// SIMATIC STEP 7 (V5.x) project Water tank
// CPU: CPU 413-2 DP
// station: Hardware
// station: SIMATIC 400(1)
// station: P_ADR_BUS
// station: P_ADR_BUS
// station: P_ADR_BUS
// station: Configuration
// program: S7 Program(1)

SYMBOL_TABLE
"Data For Temp"	DB 1	DB 1
"Temperature scaling"	FC 1	FC 1
"Motor operation"	FC 2	FC 2
"SCALE"	FC 105	FC 105	// Scaling Values
"Temp scaling"	OB 1	OB 1
"Tank-1"	PIW 256	INT	// temp for tank-1
"Tank-2"	PIW 258	INT	// temp for tank-2
"Temp-2"	PIW 512	INT	// Temp for tank 2
"Temp-1"	PIW 528	INT	// Temp for tank 1
"cooling Motor"	Q 0.0	BOOL	// water tank-1
END_SYMBOL_TABLE

FUNCTION "Temperature scaling" : WORD	// FC 1
VERSION : 0.1
VAR_OUTPUT
  RET_VAL : WORD ;
END_VAR
BEGIN
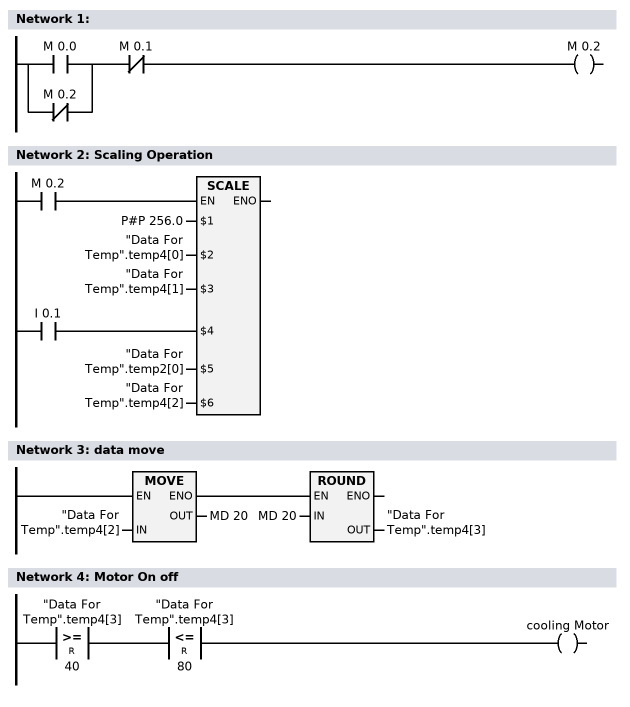
NETWORK
TITLE =
      A(;
      O     M 0.0;
      ON    M 0.2;
      );
      AN    M 0.1;
      =     M 0.2;
NETWORK
TITLE = Scaling Operation
      A     I 0.1;
      =     L 0.0;
      BLD   103;
      A     M 0.2;
      JNB   _001;
      CALL  "SCALE" (
           $1                       := P#P 256.0,
           $2                       := "Data For Temp".temp4[0],
           $3                       := "Data For Temp".temp4[1],
           $4                       := L 0.0,
           $5                       := "Data For Temp".temp2[0],
           $6                       := "Data For Temp".temp4[2]);
_001: NOP   0;
NETWORK
TITLE = data move
      A(;
      L     "Data For Temp".temp4[2];
      T     MD 20;
      SET;
      SAVE;
      CLR;
      A     BR;
      );
      JNB   _002;
      L     MD 20;
      RND;
      T     "Data For Temp".temp4[3];
_002: NOP   0;
NETWORK
TITLE = Motor On off
      A(;
      L     "Data For Temp".temp4[3];
      L     40;
      >=R;
      );
      A(;
      L     "Data For Temp".temp4[3];
      L     80;
      <=R;
      );
      =     "cooling Motor";
END_FUNCTION

// FC 105: know-how protected block, not included

DATA_BLOCK "Data For Temp"	// DB 1
VERSION : 0.1
  STRUCT
   temp : ARRAY  [0 .. 10 ] OF //Temporary placeholder variable
   BOOL  := FALSE;
   temp2 : ARRAY  [0 .. 10 ] OF WORD ;
   temp3 : ARRAY  [0 .. 10 ] OF INT ;
   temp4 : ARRAY  [0 .. 10 ] OF REAL ;
  END_STRUCT ;	
BEGIN
   temp4[0] := 1.000000e+02;
END_DATA_BLOCK

ORGANIZATION_BLOCK "Temp scaling"	// OB 1
TITLE = "Main Program Sweep (Cycle)"
VERSION : 0.1
VAR_TEMP
  OB1_EV_CLASS : BYTE ;	//Bits 0-3 = 1 (Coming event), Bits 4-7 = 1 (Event class 1)
  OB1_SCAN_1 : BYTE ;	//1 (Cold restart scan 1 of OB 1), 3 (Scan 2-n of OB 1)
  OB1_PRIORITY : BYTE ;	//Priority of OB Execution
  OB1_OB_NUMBR : BYTE ;	//1 (Organization block 1, OB1)
  OB1_RESERVED_1 : BYTE ;	//Reserved for system
  OB1_RESERVED_2 : BYTE ;	//Reserved for system
  OB1_PREV_CYCLE : INT ;	//Cycle time of previous OB1 scan (milliseconds)
  OB1_MIN_CYCLE : INT ;	//Minimum cycle time of OB1 (milliseconds)
  OB1_MAX_CYCLE : INT ;	//Maximum cycle time of OB1 (milliseconds)
  OB1_DATE_TIME : DATE_AND_TIME ;	//Date and time OB1 started
END_VAR
BEGIN
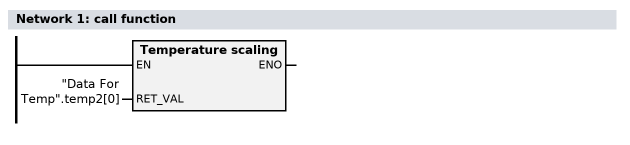
NETWORK
TITLE = call function
      CALL  "Temperature scaling" (
           RET_VAL                  := "Data For Temp".temp2[0]);
      NOP   0;
END_ORGANIZATION_BLOCK
